{attribute 'TcGenerated'}
{attribute 'no-analysis'}
{attribute 'linkalways'}
// This function has been automatically generated from the project information.
VAR_GLOBAL CONSTANT
	{attribute 'const_non_replaced'}
	stLibVersion_Project_Logic_1 : ST_LibVersion := (iMajor := 0, iMinor := 1, iBuild := 0, iRevision := 1, nFlags := 0, sVersion := '0.1.0.1');
END_VAR

(* stored: Version 1.1.0.1, ProductVersion 3.1.4024.16
   GVL Global_Version: Id {80e85591-2938-435d-a099-35507347b4d4} *)
